// TIA Portal V18 export
VAR_GLOBAL   // PLC tag table "04_5 Costanti Nomi Attuatore Stz05"
END_VAR
VAR_GLOBAL CONSTANT   // user constants
   M141 : Int := 1;   // Motore Raddrizzatrice
   P501 : Int := 2;   // EV Salita discesa rullo raddrizzatrice
END_VAR
